FUNCTION_BLOCK SM_LinearPositionMeasurementU32
VAR_INPUT
	///Measured raw value
	{attribute 'OPC.UA.DA' := '0'}
	rawValue AT %I*: UDINT;
	///Error
	{attribute 'OPC.UA.DA' := '0'}
	error AT %I*: BOOL;
	///Underrange
	{attribute 'OPC.UA.DA' := '0'}
	underrange AT %I*: BOOL;
	///Overrange
	{attribute 'OPC.UA.DA' := '0'}
	overrange AT %I*: BOOL;
	///rawValue * conversionFactor = millimeters.value
	{attribute 'OPC.UA.DA' := '0'}
	conversionFactor: LREAL := 4.65661287525E-10;
END_VAR
VAR_OUTPUT
	///Current status description
	{attribute 'OPC.UA.DA' := '1'}
	{attribute 'OPC.UA.DA.Access' := '1'}
	actualStatus: STRING;
	///Actual value
	{attribute 'OPC.UA.DA' := '1'}
	{attribute 'OPC.UA.DA.Access' := '1'}
	actual: LinearPosition;
	///Moving average value
	{attribute 'OPC.UA.DA' := '1'}
	{attribute 'OPC.UA.DA.Access' := '1'}
	average: LinearPosition;
	///Statuses of the state machine
	statuses: LinearPositionMeasurementU32Statuses;
END_VAR
VAR_IN_OUT
	///Reference to the config (alarms in millimeters)
	{attribute 'OPC.UA.DA' := '0'}
	config: MeasurementConfig;
END_VAR
VAR
END_VAR

actual( newMillimetersValue := (rawValue * conversionFactor) + config.offset );
statuses.enabledStatus( isEnabled := config.enabled );
statuses.healthStatus(
    superState := statuses.enabledStatus.enabled,
    isGood := NOT(error OR (underrange OR (overrange OR (statuses.alarmStatus.hiHi OR statuses.alarmStatus.loLo)))),
    hasWarning := statuses.alarmStatus.hi OR statuses.alarmStatus.lo);
statuses.alarmStatus(
    superState := statuses.enabledStatus.enabled,
    config := config.alarms,
    value := average.millimeters.value);

END_FUNCTION_BLOCK

(* stored: Version 1.1.0.1, ProductVersion 3.1.4019.2
   POU SM_LinearPositionMeasurementU32: Id {08b60f46-96c3-4bec-9df6-ea0161c31b6d}, SpecialFunc None *)
